Omron CX-Programmer project NewProject (CX-Programmer 9.61)

# PLC NewPLC1: CP1H XA

## Global symbols (name address type ; comment)
0.00 BOOL  ; START
0.01 BOOL  ; STOP
100.00 BOOL  ; VALVE1
100.01 BOOL  ; MOTOR
100.02 BOOL  ; MIXER
100.03 BOOL  ; VALVE2
T0000 BOOL  ; TIM1
T0001 BOOL  ; TIM2
T0002 BOOL  ; TIM3

## Program NewProgram1 (cyclic task 0)

### Section Section1

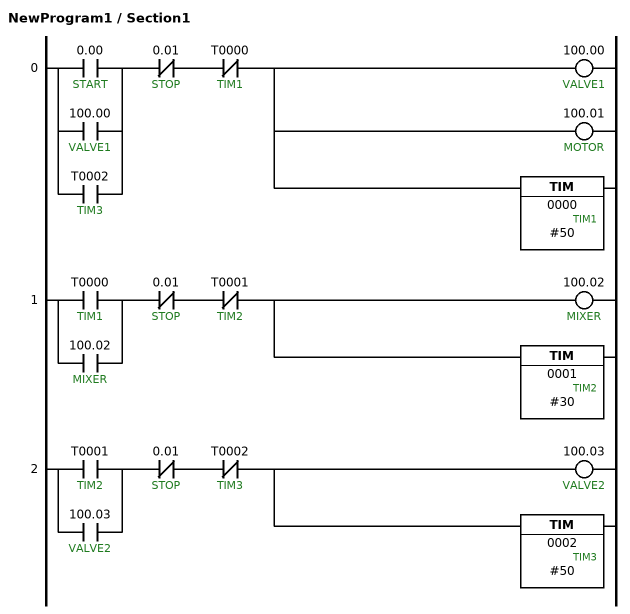
; rung 0
LD 0.00  ; START
OR 100.00  ; VALVE1
OR T0002  ; TIM3
ANDNOT 0.01  ; STOP
ANDNOT T0000  ; TIM1
OUT 100.00  ; VALVE1
OUT 100.01  ; MOTOR
TIM 0000 #50  ; TIM1
; rung 1
LD T0000  ; TIM1
OR 100.02  ; MIXER
ANDNOT 0.01  ; STOP
ANDNOT T0001  ; TIM2
OUT 100.02  ; MIXER
TIM 0001 #30  ; TIM2
; rung 2
LD T0001  ; TIM2
OR 100.03  ; VALVE2
ANDNOT 0.01  ; STOP
ANDNOT T0002  ; TIM3
OUT 100.03  ; VALVE2
TIM 0002 #50  ; TIM3

### Section END
; rung 0
END(001)